# EPICS substitutions: SemBuilder/iocs/BL99I-LCH-IOC-01/BL99I-LCH-IOC-01App/Db/BL99I-LCH-IOC-01_expanded.substitutions
# This file was automatically generated on Thu 06 Dec 2018 14:59:37 GMT from
# source: /home/jjc62351/work/Builder/SemBuilder/etc/makeIocs/BL99I-LCH-IOC-01.xml
#
# *** Please do not edit this file: edit the source file instead. ***
#

# Macros:
#  P        Device Prefix
#  PORT     Asyn Port name
#  TIMEOUT  Timeout
#  ADDR     Asyn Port address
file $(ADJEOL_JSM_IT100)/db/ADJeol.db
{
pattern { P, PORT, TIMEOUT, ADDR }
    { "BL99I-LCH-SEM-01", "semPort", "1", "0" }
}
